TEXTLIST nDriveEventTableHeader
  0 = 'Eksen' | English: 'Axis ID' | Turkish: 'Eksen'
  1 = 'Diag Kodu' | English: 'Diag Number' | Turkish: 'Diag Kodu'
  2 = 'Diag Mesaji' | English: 'Diag Message' | Turkish: 'Diag Mesaji'
  3 = 'Zaman' | English: 'Event Time' | Turkish: 'Zaman'
   = ''
END_TEXTLIST

(* stored: Version 1.1.0.1, ProductVersion 3.1.4024.6
   TextList nDriveEventTableHeader: Id {00f0e61c-1b76-459d-9f12-f4968b3556e1} *)
